	30: // Parse results
		_intRet := STRING_TO_INT(_inst_strRet);
		IF _intRet > 0 THEN
			_bResult := TRUE;
			THIS^.M_LogMessage(_strEND_MSG);
			// DO ANY PARSING HERE
			bConnected := TRUE;
		// Set error if command failed
		ELSE
			THIS^.M_SetError(_udintERROR_ID, _strERROR_MSG);
		END_IF
		// Go back to start
		_inst_intStep := 0;
END_CASE
M_StartMarking := _bResult;
intMStartMarkingStep := _inst_intStep;
END_METHOD

METHOD PUBLIC M_StopMarking : BOOL
VAR_INPUT
END_VAR

VAR CONSTANT
	_strCOMMAND_NAME : T_MaxString	:= 'StopMarking'; // Name of the API method
	_timeCOMMAND_TIMEOUT : TIME		:= T#30S; // Max time to receive API response
	_strSTART_MSG : T_MaxString		:= 'StoppingMarking'; // Prints when method starts
	_strEND_MSG : T_MaxString		:= 'StoppedMarking'; // Prints when method finishes
	_udintERROR_ID : UDINT			:= KeyenceLaserMarkerMDX2000_Error.FailedToStopMarking; // Error ID to set if command fails
	_strERROR_MSG : T_MaxString		:= 'Failed to Stop Marking by Laser Marker!'; // Error message to set if command fails
END_VAR

VAR_INST
	_inst_arrParams: T_ApiParameterList; // Parameters array
	_inst_arrOutputs: T_ApiParameterList; // Outputs array
	_inst_strRet: T_ApiParamValue; // Return string from the router
	_inst_intStep: INT; // Current method step
	_inst_fbParams: FB_ApiParamBuilder; // Parameter builder FB
END_VAR

VAR
	_bComplete: BOOL; // True if the routing finishes
	_intRet: INT; // Return string converted to an integer
	_bResult : BOOL; // Output of the method
END_VAR
_bResult := FALSE;
bMStopMarkingBusy := TRUE;
_inst_intStep := intMStopMarkingStep;
CASE _inst_intStep OF
	0: // Wait for no error and router not busy
		IF NOT THIS^.P_bError AND NOT bRouterBusy THEN
			bRouterBusy := TRUE;
			_inst_intStep := _inst_intStep + 10;
		END_IF
		
	10: // Initialize parameters
		THIS^.M_LogMessage(_strSTART_MSG);
		_inst_fbParams.M_ClearParameters();
		// ADD ANY PARAMETERS HERE
		_inst_fbParams.M_OutputToParameterList(_inst_arrParams);
		_inst_intStep := _inst_intStep + 10;
		
	20: // Route the command
		_bComplete := M_RouterHelper(
			_in_strMethodName := _strCOMMAND_NAME, 
			_in_timeTimeout := _timeCOMMAND_TIMEOUT,
			_inout_arrParams := _inst_arrParams,
			_inout_arrOutputs := _inst_arrOutputs,
			_out_strReturnValue=>_inst_strRet);
		
		// If route completed, move to next step
		IF _bComplete THEN
			_inst_intStep := _inst_intStep + 10;
			bRouterBusy := FALSE;
		ELSIF THIS^.P_bError THEN
			_inst_intStep := 0;
			bRouterBusy := FALSE;
		END_IF
		
	30: // Parse results
		_intRet := STRING_TO_INT(_inst_strRet);
		IF _intRet > 0 THEN
			_bResult := TRUE;
			THIS^.M_LogMessage(_strEND_MSG);
			// DO ANY PARSING HERE
			bConnected := TRUE;
		// Set error if command failed
		ELSE
			THIS^.M_SetError(_udintERROR_ID, _strERROR_MSG);
		END_IF
		// Go back to start
		_inst_intStep := 0;
END_CASE
M_StopMarking := _bResult;
intMStopMarkingStep := _inst_intStep;
END_METHOD

METHOD M_UpdateAllMarkingInformation : BOOL
VAR_INPUT
	MaxNumberOfBlocks	: INT;
//	MarkingInfo_Array	: ARRAY [0..255] OF OneBlockInfo;
END_VAR

VAR CONSTANT
	_strCOMMAND_NAME : T_MaxString	:= 'UpdateAllMarkingInformation'; // Name of the API method
	_timeCOMMAND_TIMEOUT : TIME		:= T#30S; // Max time to receive API response
	_strSTART_MSG : T_MaxString		:= 'UpdatingAllMarkingInformationInTheLaserProgram'; // Prints when method starts
	_strEND_MSG : T_MaxString		:= 'UpdatedAllMarkingInformationInTheLaserProgram'; // Prints when method finishes
	_udintERROR_ID : UDINT			:= KeyenceLaserMarkerMDX2000_Error.FailedToUpdateAllMarkingInformation; // Error ID to set if command fails
	_strERROR_MSG : T_MaxString		:= 'Failed to update All Marking Information in the Laser Marker program!'; // Error message to set if command fails
END_VAR

VAR_INST
	_inst_arrParams: T_ApiParameterList; // Parameters array
	_inst_arrOutputs: T_ApiParameterList; // Outputs array
	_inst_strRet: T_ApiParamValue; // Return string from the router
	_inst_intStep: INT; // Current method step
	_inst_fbParams: FB_ApiParamBuilder; // Parameter builder FB
END_VAR

VAR
	_bComplete: BOOL; // True if the routing finishes
	_intRet: INT; // Return string converted to an integer
	_bResult : BOOL; // Output of the method
	intIndex: INT;
	intIndex2 : INT;
	bOneTimeOnly : BOOL := TRUE;
END_VAR
_bResult := FALSE;
bMUpdateAllMarkingInfoBusy := TRUE;
_inst_intStep := intMUpdateAllMarkingInfoStep;
CASE _inst_intStep OF
	0: // Wait for no error and router not busy
		IF NOT THIS^.P_bError AND NOT bRouterBusy THEN
			bRouterBusy := TRUE;
			_inst_intStep := _inst_intStep + 10;
		END_IF
		
	10: // Initialize parameters
		THIS^.M_LogMessage(_strSTART_MSG);
		_inst_fbParams.M_ClearParameters();
		// ADD ANY PARAMETERS HERE
		_inst_fbParams.M_AddParameter('MaxNumberOfBlocks', MaxNumberOfBlocks);
		_inst_fbParams.M_OutputToParameterList(_inst_arrParams);
		_inst_intStep := _inst_intStep + 10;
		
	20: // Route the command
		_bComplete := M_RouterHelper(
			_in_strMethodName := _strCOMMAND_NAME, 
			_in_timeTimeout := _timeCOMMAND_TIMEOUT,
			_inout_arrParams := _inst_arrParams,
			_inout_arrOutputs := _inst_arrOutputs,
			_out_strReturnValue=>_inst_strRet);
		
		// If route completed, move to next step
		IF _bComplete THEN
			_inst_intStep := _inst_intStep + 10;
			bRouterBusy := FALSE;
		ELSIF THIS^.P_bError THEN
			_inst_intStep := 0;
			bRouterBusy := FALSE;
		END_IF
		
	30: // Parse results
		_intRet := STRING_TO_INT(_inst_strRet);
		IF _intRet > 0 THEN
			_bResult := TRUE;
			THIS^.M_LogMessage(_strEND_MSG);
			// DO ANY PARSING HERE
			_inst_fbParams.M_LoadFromParameterList(_inst_arrOutputs);
			bConnected := TRUE;
		// Set error if command failed
		ELSE
			THIS^.M_SetError(_udintERROR_ID, _strERROR_MSG);
		END_IF
		// Go back to start
		_inst_intStep := 0;
END_CASE
M_UpdateAllMarkingInformation := _bResult;
intMUpdateAllMarkingInfoStep := _inst_intStep;
END_METHOD

METHOD PUBLIC M_UpdateSingleBlockMarkingInformation : BOOL
VAR_INPUT
	BlockNumber : INT;
	BlockData : STRING;
	MarkEnabled : BOOL;
END_VAR

VAR CONSTANT
	_strCOMMAND_NAME : T_MaxString	:= 'UpdateSingleBlockMarkingInformation'; // Name of the API method
	_timeCOMMAND_TIMEOUT : TIME		:= T#30S; // Max time to receive API response
	_strSTART_MSG : T_MaxString		:= 'UpdatingSingleBlockMarkingInformationInTheLaserProgram'; // Prints when method starts
	_strEND_MSG : T_MaxString		:= 'UpdatedSingleBlockMarkingInformationInTheLaserProgram'; // Prints when method finishes
	_udintERROR_ID : UDINT			:= KeyenceLaserMarkerMDX2000_Error.FailedToUpdateSingleBlockMarkingInformation; // Error ID to set if command fails
	_strERROR_MSG : T_MaxString		:= 'Failed to update single block Marking Information in the Laser Marker program!'; // Error message to set if command fails
END_VAR

VAR_INST
	_inst_arrParams: T_ApiParameterList; // Parameters array
	_inst_arrOutputs: T_ApiParameterList; // Outputs array
	_inst_strRet: T_ApiParamValue; // Return string from the router
	_inst_intStep: INT; // Current method step
	_inst_fbParams: FB_ApiParamBuilder; // Parameter builder FB
END_VAR

VAR
	_bComplete: BOOL; // True if the routing finishes
	_intRet: INT; // Return string converted to an integer
	_bResult : BOOL; // Output of the method
	BlockType_INT : INT;
END_VAR
_bResult := FALSE;
bMUpdateSingleBlockInfoBusy := TRUE;
_inst_intStep := intMUpdateSingleBlockInfoStep;
CASE _inst_intStep OF
	0: // Wait for no error and router not busy
		IF NOT THIS^.P_bError AND NOT bRouterBusy THEN
			bRouterBusy := TRUE;
			_inst_intStep := _inst_intStep + 10;
		END_IF
		
	10: // Initialize parameters
		THIS^.M_LogMessage(_strSTART_MSG);
		_inst_fbParams.M_ClearParameters();
		// ADD ANY PARAMETERS HERE
		_inst_fbParams.M_AddParameter('BlockNumber', BlockNumber);
		_inst_fbParams.M_AddParameter('BlockData', BlockData);
		_inst_fbParams.M_AddParameter('MarkEnabled', MarkEnabled);
		_inst_fbParams.M_OutputToParameterList(_inst_arrParams);
		_inst_intStep := _inst_intStep + 10;
		
	20: // Route the command
		_bComplete := M_RouterHelper(
			_in_strMethodName := _strCOMMAND_NAME, 
			_in_timeTimeout := _timeCOMMAND_TIMEOUT,
			_inout_arrParams := _inst_arrParams,
			_inout_arrOutputs := _inst_arrOutputs,
			_out_strReturnValue=>_inst_strRet);
		
		// If route completed, move to next step
		IF _bComplete THEN
			_inst_intStep := _inst_intStep + 10;
			bRouterBusy := FALSE;
		ELSIF THIS^.P_bError THEN
			_inst_intStep := 0;
			bRouterBusy := FALSE;
		END_IF
		
	30: // Parse results
		_intRet := STRING_TO_INT(_inst_strRet);
		IF _intRet > 0 THEN
			_bResult := TRUE;
			THIS^.M_LogMessage(_strEND_MSG);
			// DO ANY PARSING HERE
			_inst_fbParams.M_LoadFromParameterList(_inst_arrOutputs);
			bConnected := TRUE;
		// Set error if command failed
		ELSE
			THIS^.M_SetError(_udintERROR_ID, _strERROR_MSG);
		END_IF
		// Go back to start
		_inst_intStep := 0;
END_CASE
M_UpdateSingleBlockMarkingInformation := _bResult;
intMUpdateSingleBlockInfoStep := _inst_intStep;
END_METHOD

(* This method should explicitly get the current program loaded on the device.
	If the current program is successfully gotten, this method should return
	TRUE and set P_strCurrentProgram and strCurrentProgram to the gotten
	program name. If this method fails, both should be set to empty strings. *)
METHOD M_GetCurrentProgram : BOOL
VAR_OUTPUT
	(* This should be set to the name of the currently loaded program if
		the method was successful, or a blank string otherwise. *)
	strCurrentProgram	: Sensata_Common.T_MaxString;
END_VAR
VAR CONSTANT
	_strCOMMAND_NAME : T_MaxString	:= 'GetCurrentProgram'; // Name of the API method
	_timeCOMMAND_TIMEOUT : TIME		:= T#45S; // Max time to receive API response
	_strSTART_MSG : T_MaxString		:= 'GettingCurrentProgramFromLaserMemory'; // Prints when method starts
	_strEND_MSG : T_MaxString		:= 'GotCurrentProgramFromLaserMemory'; // Prints when method finishes
	_udintERROR_ID : UDINT			:= KeyenceLaserMarkerMDX2000_Error.FailedToGetCurrentProgram; // Error ID to set if command fails
	_strERROR_MSG : T_MaxString		:= 'Failed to Get Current Laser Program from Laser Marker!'; // Error message to set if command fails
END_VAR

VAR_INST
	_inst_arrParams: T_ApiParameterList; // Parameters array
	_inst_arrOutputs: T_ApiParameterList; // Outputs array
	_inst_strRet: T_ApiParamValue; // Return string from the router
	_inst_intStep: INT; // Current method step
	_inst_fbParams: FB_ApiParamBuilder; // Parameter builder FB
END_VAR

VAR
	_bComplete: BOOL; // True if the routing finishes
	_intRet: INT; // Return string converted to an integer
	_bResult : BOOL; // Output of the method
END_VAR
_bResult := FALSE;
bMGetCurrentProgBusy := TRUE;
_inst_intStep := intMGetCurrentProgStep;
CASE _inst_intStep OF
	0: // Wait for no error and router not busy
		IF NOT THIS^.P_bError AND NOT bRouterBusy THEN
			bRouterBusy := TRUE;
			_inst_intStep := _inst_intStep + 10;
		END_IF
		
	10: // Initialize parameters
		THIS^.M_LogMessage(_strSTART_MSG);
		_inst_fbParams.M_ClearParameters();
		// ADD ANY PARAMETERS HERE
		_inst_fbParams.M_OutputToParameterList(_inst_arrParams);
		_inst_intStep := _inst_intStep + 10;
		
	20: // Route the command
		_bComplete := M_RouterHelper(
			_in_strMethodName := _strCOMMAND_NAME, 
			_in_timeTimeout := _timeCOMMAND_TIMEOUT,
			_inout_arrParams := _inst_arrParams,
			_inout_arrOutputs := _inst_arrOutputs,
			_out_strReturnValue=>_inst_strRet);
		
		// If route completed, move to next step
		IF _bComplete THEN
			_inst_intStep := _inst_intStep + 10;
			bRouterBusy := FALSE;
		ELSIF THIS^.P_bError THEN
			_inst_intStep := 0;
			bRouterBusy := FALSE;
		END_IF
		
	30: // Parse results
		_intRet := STRING_TO_INT(_inst_strRet);
		IF _intRet > 0 THEN
			_bResult := TRUE;
			THIS^.M_LogMessage(_strEND_MSG);
			// DO ANY PARSING HERE
			_inst_fbParams.M_LoadFromParameterList(_inst_arrOutputs);
			strCurrentProgram := _inst_fbParams.M_ParseString(_inst_fbParams.M_GetParameter('programName'));
			bConnected := TRUE;
		// Set error if command failed
		ELSE
			THIS^.M_SetError(_udintERROR_ID, _strERROR_MSG);
		END_IF
		// Go back to start
		_inst_intStep := 0;
END_CASE
M_GetCurrentProgram := _bResult;
intMGetCurrentProgStep := _inst_intStep;
END_METHOD

(* This method should explicitly check the program state of the device.
	Once the program state is known, this method should return TRUE and set
	P_enumProgramState and enumProgramState to the relevant E_ProgramState
	value, else it should set both to E_ProgramState.Unknown. *)
METHOD M_GetProgramState : BOOL
VAR_OUTPUT
	(* If the program state is successfully gotten, this should be set to
		the relevant E_ProgramState value. If this method fails, this should
		be set to E_ProgramState.Unknown. *)
	enumProgramState	: Sensata_Common.E_ProgramState;
END_VAR
M_GetProgramState := TRUE;
THIS^.M_LogWarning('M_GetProgramState is not implemented!');
END_METHOD

(* This method should load a new program onto the device, and then return TRUE
	once program loading is completed. Once this method begins the program loading
	process, P_strCurrentProgram should be cleared unless it is still explicitly
	known to be loaded. *)
METHOD M_LoadProgram : BOOL
VAR_INPUT
	(* String representing the program to load. If string must be in a specific
		format, make sure to override this comment to document it. *)
	//strProgram	: Sensata_Common.T_MaxString;
	
	//Replace filepath with just program number and also 
//	filepath : STRING;	// filepath where the program is stored
//	LaserMemoryLocation : INT; // Laser Memory location where the program needs to be loaded 
	
END_VAR

VAR CONSTANT
	_strCOMMAND_NAME : T_MaxString	:= 'LoadProgram'; // Name of the API method
	_timeCOMMAND_TIMEOUT : TIME		:= T#30S; // Max time to receive API response
	_strSTART_MSG : T_MaxString		:= 'LoadingProgramToLaser'; // Prints when method starts
	_strEND_MSG : T_MaxString		:= 'ProgramLoadedToLaser'; // Prints when method finishes
	_udintERROR_ID : UDINT			:= KeyenceLaserMarkerMDX2000_Error.FailedToSendProgramToLaser; // Error ID to set if command fails
	_strERROR_MSG : T_MaxString		:= 'Failed to Load Program to Laser Marker!'; // Error message to set if command fails
END_VAR

VAR_INST
	_inst_arrParams: T_ApiParameterList; // Parameters array
	_inst_arrOutputs: T_ApiParameterList; // Outputs array
	_inst_strRet: T_ApiParamValue; // Return string from the router
	_inst_intStep: INT; // Current method step
	_inst_fbParams: FB_ApiParamBuilder; // Parameter builder FB
END_VAR

VAR
	_bComplete: BOOL; // True if the routing finishes
	_intRet: INT; // Return string converted to an integer
	_bResult : BOOL; // Output of the method	
END_VAR
_bResult := FALSE;
bMLoadProgramBusy := TRUE;
_inst_intStep := intMLoadProgramStep;
CASE _inst_intStep OF
	0: // Wait for no error and router not busy
		IF NOT THIS^.P_bError AND NOT bRouterBusy THEN
			bRouterBusy := TRUE;
			_inst_intStep := _inst_intStep + 10;
		END_IF
		
	10: // Initialize parameters
		THIS^.M_LogMessage(_strSTART_MSG);
		_inst_fbParams.M_ClearParameters();
		// ADD ANY PARAMETERS HERE
		_inst_fbParams.M_AddParameter('programName', in_strProgram);
		_inst_fbParams.M_OutputToParameterList(_inst_arrParams);
		_inst_intStep := _inst_intStep + 10;
		
	20: // Route the command
		_bComplete := M_RouterHelper(
			_in_strMethodName := _strCOMMAND_NAME, 
			_in_timeTimeout := _timeCOMMAND_TIMEOUT,
			_inout_arrParams := _inst_arrParams,
			_inout_arrOutputs := _inst_arrOutputs,
			_out_strReturnValue=>_inst_strRet);
		
		// If route completed, move to next step
		IF _bComplete THEN
			_inst_intStep := _inst_intStep + 10;
			bRouterBusy := FALSE;
		ELSIF THIS^.P_bError THEN
			_inst_intStep := 0;
			bRouterBusy := FALSE;
		END_IF
		
	30: // Parse results
		_intRet := STRING_TO_INT(_inst_strRet);
		IF _intRet > 0 THEN
			_bResult := TRUE;
			THIS^.M_LogMessage(_strEND_MSG);
			// DO ANY PARSING HERE
		// Set error if command failed
		ELSE
			THIS^.M_SetError(_udintERROR_ID, _strERROR_MSG);
		END_IF
		// Go back to start
		_inst_intStep := 0;
END_CASE
M_LoadProgram := _bResult;
intMLoadProgramStep := _inst_intStep;
END_METHOD

(* This program should move to the program state from whatever state it was in
	to the Paused state, and then return TRUE once successful. If the program
	state is Stopped, this method should return TRUE but keep the current state
	as Stopped, since Paused at the beginning at the program is equivalent to
	being Stopped. *)
METHOD M_PauseProgram : BOOL
M_PauseProgram := TRUE;
THIS^.M_LogWarning('M_PauseProgram is not implemented!');
END_METHOD

METHOD PUBLIC M_SaveCurrentLaserProgramtoPC : BOOL
VAR_INPUT
	LaserProgramFolderPath : STRING;
END_VAR
VAR_OUTPUT
	out_bool_SaveProgramToPC_Success : BOOL;
END_VAR
VAR CONSTANT
	_strCOMMAND_NAME : T_MaxString	:= 'SaveCurrentLaserProgramToPC'; // Name of the API method
	_timeCOMMAND_TIMEOUT : TIME		:= T#45S; // Max time to receive API response
	_strSTART_MSG : T_MaxString		:= 'SavingCurrentProgram'; // Prints when method starts
	_strEND_MSG : T_MaxString		:= 'SavedCurrentProgram'; // Prints when method finishes
	_udintERROR_ID : UDINT			:= KeyenceLaserMarkerMDX2000_Error.FailedToSaveCurrentLaserProgramToPC; // Error ID to set if command fails
	_strERROR_MSG : T_MaxString		:= 'Failed to Save Current Laser Program to PC from Laser Marker!'; // Error message to set if command fails
END_VAR

VAR_INST
	_inst_arrParams: T_ApiParameterList; // Parameters array
	_inst_arrOutputs: T_ApiParameterList; // Outputs array
	_inst_strRet: T_ApiParamValue; // Return string from the router
	_inst_intStep: INT; // Current method step
	_inst_fbParams: FB_ApiParamBuilder; // Parameter builder FB
END_VAR

VAR
	_bComplete: BOOL; // True if the routing finishes
	_intRet: INT; // Return string converted to an integer
	_bResult : BOOL; // Output of the method
END_VAR
_bResult := FALSE;
bMSaveCurrentLaserProgramtoPCBusy := TRUE;
_inst_intStep := intMSaveCurrentLaserProgramtoPC;
CASE _inst_intStep OF
	0: // Wait for no error and router not busy
		IF NOT THIS^.P_bError AND NOT bRouterBusy THEN
			bRouterBusy := TRUE;
			_inst_intStep := _inst_intStep + 10;
		END_IF
		
	10: // Initialize parameters
		THIS^.M_LogMessage(_strSTART_MSG);
		_inst_fbParams.M_ClearParameters();
		// ADD ANY PARAMETERS HERE
		_inst_fbParams.M_AddParameter('LaserProgramFolderPath',LaserProgramFolderPath);
		_inst_fbParams.M_OutputToParameterList(_inst_arrParams);
		_inst_intStep := _inst_intStep + 10;
		
	20: // Route the command
		_bComplete := M_RouterHelper(
			_in_strMethodName := _strCOMMAND_NAME, 
			_in_timeTimeout := _timeCOMMAND_TIMEOUT,
			_inout_arrParams := _inst_arrParams,
			_inout_arrOutputs := _inst_arrOutputs,
			_out_strReturnValue=>_inst_strRet);
		
		// If route completed, move to next step
		IF _bComplete THEN
			_inst_intStep := _inst_intStep + 10;
			bRouterBusy := FALSE;
		ELSIF THIS^.P_bError THEN
			_inst_intStep := 0;
			bRouterBusy := FALSE;
		END_IF
		
	30: // Parse results
		_intRet := STRING_TO_INT(_inst_strRet);
		IF _intRet > 0 THEN
			_bResult := TRUE;
			THIS^.M_LogMessage(_strEND_MSG);
			// DO ANY PARSING HERE
			_inst_fbParams.M_LoadFromParameterList(_inst_arrOutputs);
			out_bool_SaveProgramToPC_Success := _inst_fbParams.M_ParseBool(_inst_fbParams.M_GetParameter('out_bool_SaveProgramToPC_Success'));
			bConnected := TRUE;
		// Set error if command failed
		ELSE
			THIS^.M_SetError(_udintERROR_ID, _strERROR_MSG);
		END_IF
		// Go back to start
		_inst_intStep := 0;
END_CASE
M_SaveCurrentLaserProgramtoPC := _bResult;
intMSaveCurrentLaserProgramtoPC := _inst_intStep;
END_METHOD

METHOD PUBLIC M_SendProgramtoLaser : BOOL
VAR_INPUT
	filepath : STRING;	// filepath where the program is stored
	LaserMemoryLocation : INT; // Laser Memory location where the program needs to be loaded 
END_VAR

VAR_OUTPUT
	out_bool_SendProgramToLaserSuccess : BOOL;
END_VAR

VAR CONSTANT
	_strCOMMAND_NAME : T_MaxString	:= 'SendProgramtoLaser'; // Name of the API method
	_timeCOMMAND_TIMEOUT : TIME		:= T#30S; // Max time to receive API response
	_strSTART_MSG : T_MaxString		:= 'SendingProgramToLaser'; // Prints when method starts
	_strEND_MSG : T_MaxString		:= 'SentProgramToLaser'; // Prints when method finishes
	_udintERROR_ID : UDINT			:= KeyenceLaserMarkerMDX2000_Error.FailedToSendProgramToLaser; // Error ID to set if command fails
	_strERROR_MSG : T_MaxString		:= 'Failed to Send Program to Laser Marker!'; // Error message to set if command fails
END_VAR

VAR_INST
	_inst_arrParams: T_ApiParameterList; // Parameters array
	_inst_arrOutputs: T_ApiParameterList; // Outputs array
	_inst_strRet: T_ApiParamValue; // Return string from the router
	_inst_intStep: INT; // Current method step
	_inst_fbParams: FB_ApiParamBuilder; // Parameter builder FB
END_VAR

VAR
	_bComplete: BOOL; // True if the routing finishes
	_intRet: INT; // Return string converted to an integer
	_bResult : BOOL; // Output of the method	

END_VAR
_bResult := FALSE;
bMSendProgramToLaserBusy := TRUE;
_inst_intStep := intMSendProgramToLaserStep;
CASE _inst_intStep OF
	0: // Wait for no error and router not busy
		IF NOT THIS^.P_bError AND NOT bRouterBusy THEN
			bRouterBusy := TRUE;
			_inst_intStep := _inst_intStep + 10;
		END_IF
		
	10: // Initialize parameters
		THIS^.M_LogMessage(_strSTART_MSG);
		_inst_fbParams.M_ClearParameters();
		// ADD ANY PARAMETERS HERE
		_inst_fbParams.M_AddParameter('filepath', filepath);
		_inst_fbParams.M_AddParameter('LaserMemoryLocation', LaserMemoryLocation);
		_inst_fbParams.M_OutputToParameterList(_inst_arrParams);
		_inst_intStep := _inst_intStep + 10;
		
	20: // Route the command
		_bComplete := M_RouterHelper(
			_in_strMethodName := _strCOMMAND_NAME, 
			_in_timeTimeout := _timeCOMMAND_TIMEOUT,
			_inout_arrParams := _inst_arrParams,
			_inout_arrOutputs := _inst_arrOutputs,
			_out_strReturnValue=>_inst_strRet);
		
		// If route completed, move to next step
		IF _bComplete THEN
			_inst_intStep := _inst_intStep + 10;
			bRouterBusy := FALSE;
		ELSIF THIS^.P_bError THEN
			_inst_intStep := 0;
			bRouterBusy := FALSE;
		END_IF
		
	30: // Parse results
		_intRet := STRING_TO_INT(_inst_strRet);
		IF _intRet > 0 THEN
			_bResult := TRUE;
			THIS^.M_LogMessage(_strEND_MSG);
			// DO ANY PARSING HERE
			_inst_fbParams.M_LoadFromParameterList(_inst_arrOutputs);
			out_bool_SendProgramToLaserSuccess := _inst_fbParams.M_ParseBool(_inst_fbParams.M_GetParameter('out_bool_SendProgramToLaserSuccess'));
			bConnected := TRUE;
		// Set error if command failed
		ELSE
			THIS^.M_SetError(_udintERROR_ID, _strERROR_MSG);
		END_IF
		// Go back to start
		_inst_intStep := 0;
END_CASE
M_SendProgramtoLaser := _bResult;
intMSendProgramToLaserStep := _inst_intStep;
END_METHOD

(* This should move the program state from whatever state it is in to the
	Running state, and then return TRUE once successful. Starting from the
	Paused state should always continue execution from whatever point the
	program was at when the program was initially paused. *)
METHOD M_StartProgram : BOOL
M_StartProgram := TRUE;
THIS^.M_LogWarning('M_StartProgram is not implemented!');
END_METHOD

(* This should change the program state from whatever state it was in to the
	Stopped state and then return TRUE. Moving to the Stopped state should
	always reset the program execution back to the beginning. *)
METHOD M_StopProgram : BOOL
M_StopProgram := TRUE;
THIS^.M_LogWarning('M_StopProgram is not implemented!');
END_METHOD

METHOD PUBLIC M_UpdateSingleProgramBlockData : BOOL
VAR_INPUT
	LaserProgramMemoryLocation : INT;
	BlockNumber : INT;
	BlockData : STRING;
	BlockType : BlockTypes;
END_VAR
VAR_OUTPUT
	out_bool_UpdateData_Success : BOOL;
END_VAR
VAR CONSTANT
	_strCOMMAND_NAME : T_MaxString	:= 'UpdateSingleBlockData'; // Name of the API method
	_timeCOMMAND_TIMEOUT : TIME		:= T#30S; // Max time to receive API response
	_strSTART_MSG : T_MaxString		:= 'UpdatingSingleBlockdataInTheLaserProgram'; // Prints when method starts
	_strEND_MSG : T_MaxString		:= 'UpdatedSingleBlockdataInTheLaserProgram'; // Prints when method finishes
	_udintERROR_ID : UDINT			:= KeyenceLaserMarkerMDX2000_Error.FailedToUpdateSingleBlockData; // Error ID to set if command fails
	_strERROR_MSG : T_MaxString		:= 'Failed to update single block data in the Laser Marker program!'; // Error message to set if command fails
END_VAR

VAR_INST
	_inst_arrParams: T_ApiParameterList; // Parameters array
	_inst_arrOutputs: T_ApiParameterList; // Outputs array
	_inst_strRet: T_ApiParamValue; // Return string from the router
	_inst_intStep: INT; // Current method step
	_inst_fbParams: FB_ApiParamBuilder; // Parameter builder FB
END_VAR

VAR
	_bComplete: BOOL; // True if the routing finishes
	_intRet: INT; // Return string converted to an integer
	_bResult : BOOL; // Output of the method
	BlockType_INT : INT;
END_VAR
_bResult := FALSE;
bMUpdateSingleProgramBlockDataBusy := TRUE;
_inst_intStep := intMUpdateSingleProgramBlockDataStep;
CASE _inst_intStep OF
	0: // Wait for no error and router not busy
		IF NOT THIS^.P_bError AND NOT bRouterBusy THEN
			bRouterBusy := TRUE;
			_inst_intStep := _inst_intStep + 10;
		END_IF
		
	10: // Initialize parameters
		THIS^.M_LogMessage(_strSTART_MSG);
		_inst_fbParams.M_ClearParameters();
		// ADD ANY PARAMETERS HERE
		BlockType_INT := TO_INT(BlockType);
		_inst_fbParams.M_AddParameter('LaserProgramMemoryLocation', LaserProgramMemoryLocation);
		_inst_fbParams.M_AddParameter('BlockNumber', BlockNumber);
		_inst_fbParams.M_AddParameter('BlockData', BlockData);
		_inst_fbParams.M_AddParameter('BlockType', BlockType_INT);
		_inst_fbParams.M_OutputToParameterList(_inst_arrParams);
		_inst_intStep := _inst_intStep + 10;
		
	20: // Route the command
		_bComplete := M_RouterHelper(
			_in_strMethodName := _strCOMMAND_NAME, 
			_in_timeTimeout := _timeCOMMAND_TIMEOUT,
			_inout_arrParams := _inst_arrParams,
			_inout_arrOutputs := _inst_arrOutputs,
			_out_strReturnValue=>_inst_strRet);
		
		// If route completed, move to next step
		IF _bComplete THEN
			_inst_intStep := _inst_intStep + 10;
			bRouterBusy := FALSE;
		ELSIF THIS^.P_bError THEN
			_inst_intStep := 0;
			bRouterBusy := FALSE;
		END_IF
		
	30: // Parse results
		_intRet := STRING_TO_INT(_inst_strRet);
		IF _intRet > 0 THEN
			_bResult := TRUE;
			THIS^.M_LogMessage(_strEND_MSG);
			// DO ANY PARSING HERE
			_inst_fbParams.M_LoadFromParameterList(_inst_arrOutputs);
			out_bool_UpdateData_Success := _inst_fbParams.M_ParseBool(_inst_fbParams.M_GetParameter('out_bool_UpdateData_Success'));
			bConnected := TRUE;
		// Set error if command failed
		ELSE
			THIS^.M_SetError(_udintERROR_ID, _strERROR_MSG);
		END_IF
		// Go back to start
		_inst_intStep := 0;
END_CASE
M_UpdateSingleProgramBlockData := _bResult;
intMUpdateSingleProgramBlockDataStep := _inst_intStep;
END_METHOD

METHOD PUBLIC M_UpdateSingleProgramBlockMarkEnabled : BOOL
VAR_INPUT
	LaserProgramMemoryLocation : INT;
	BlockNumber : INT;
	BlockType : BlockTypes;
	MarkEnabled : BOOL;
	//int LaserProgramMemoryLocation, int BlockNumber, bool MarkEnabled, BlockTypes BlockType, out bool out_bool_UpdateSingleBlockMarkEnabledIntheLaser_Success
END_VAR
VAR_OUTPUT
	out_bool_MarkEnabled_Success : BOOL;
END_VAR
VAR CONSTANT
	_strCOMMAND_NAME : T_MaxString	:= 'UpdateSingleBlockMarkEnabled'; // Name of the API method
	_timeCOMMAND_TIMEOUT : TIME		:= T#30S; // Max time to receive API response
	_strSTART_MSG : T_MaxString		:= 'UpdatingSingleBlockMarkEnabledStatusInTheLaserProgram'; // Prints when method starts
	_strEND_MSG : T_MaxString		:= 'UpdatedSingleBlockMarkEnabledStatusInTheLaserProgram'; // Prints when method finishes
	_udintERROR_ID : UDINT			:= KeyenceLaserMarkerMDX2000_Error.FailedToUpdateSingleBlockMarkEnabledProperty; // Error ID to set if command fails
	_strERROR_MSG : T_MaxString		:= 'Failed to update single block mark enabled status in the Laser Marker program!'; // Error message to set if command fails
END_VAR

VAR_INST
	_inst_arrParams: T_ApiParameterList; // Parameters array
	_inst_arrOutputs: T_ApiParameterList; // Outputs array
	_inst_strRet: T_ApiParamValue; // Return string from the router
	_inst_intStep: INT; // Current method step
	_inst_fbParams: FB_ApiParamBuilder; // Parameter builder FB
END_VAR

VAR
	_bComplete: BOOL; // True if the routing finishes
	_intRet: INT; // Return string converted to an integer
	_bResult : BOOL; // Output of the method
	_dummy_pointer : PVOID;
	BlockType_INT : INT;
END_VAR
_bResult := FALSE;
bMUpdateSingleProgramBlockMarkingEnabledBusy := TRUE;
_inst_intStep := intMUpdateSingleProgramBlockMarkingEnabledStep;
CASE _inst_intStep OF
	0: // Wait for no error and router not busy
		IF NOT THIS^.P_bError AND NOT bRouterBusy THEN
			bRouterBusy := TRUE;
			_inst_intStep := _inst_intStep + 10;
		END_IF
		
	10: // Initialize parameters
		THIS^.M_LogMessage(_strSTART_MSG);
		_inst_fbParams.M_ClearParameters();
		// ADD ANY PARAMETERS HERE
		BlockType_INT := TO_INT(BlockType);
		_inst_fbParams.M_AddParameter('LaserProgramMemoryLocation', LaserProgramMemoryLocation);
		_inst_fbParams.M_AddParameter('BlockNumber', BlockNumber);
		_inst_fbParams.M_AddParameter('MarkEnabled', MarkEnabled);
		_inst_fbParams.M_AddParameter('BlockType', BlockType_INT);
		_inst_fbParams.M_OutputToParameterList(_inst_arrParams);
		_inst_intStep := _inst_intStep + 10;
		
	20: // Route the command
		_bComplete := M_RouterHelper(
			_in_strMethodName := _strCOMMAND_NAME, 
			_in_timeTimeout := _timeCOMMAND_TIMEOUT,
			_inout_arrParams := _inst_arrParams,
			_inout_arrOutputs := _inst_arrOutputs,
			_out_strReturnValue=>_inst_strRet);
		
		// If route completed, move to next step
		IF _bComplete THEN
			_inst_intStep := _inst_intStep + 10;
			bRouterBusy := FALSE;
		ELSIF THIS^.P_bError THEN
			_inst_intStep := 0;
			bRouterBusy := FALSE;
		END_IF
		
	30: // Parse results
		_intRet := STRING_TO_INT(_inst_strRet);
		IF _intRet > 0 THEN
			_bResult := TRUE;
			THIS^.M_LogMessage(_strEND_MSG);
			// DO ANY PARSING HERE
			_inst_fbParams.M_LoadFromParameterList(_inst_arrOutputs);
			out_bool_MarkEnabled_Success := _inst_fbParams.M_ParseBool(_inst_fbParams.M_GetParameter('out_bool_MarkEnabled_Success'));
			bConnected := TRUE;
		// Set error if command failed
		ELSE
			THIS^.M_SetError(_udintERROR_ID, _strERROR_MSG);
		END_IF
		// Go back to start
		_inst_intStep := 0;
END_CASE
M_UpdateSingleProgramBlockMarkEnabled := _bResult;
intMUpdateSingleProgramBlockMarkingEnabledStep := _inst_intStep;
END_METHOD

(* This property should be TRUE while any method in this interface is actively
	executing, or FALSE otherwise. *)
PROPERTY P_bProgramControlBusy : BOOL
GET
END_GET
END_PROPERTY

(* The current E_ProgramState value of the device. This should be reset to
	E_ProgramState.Unknown if any methods in this interface interact with the
	device but fail. *)
PROPERTY P_enumProgramState : Sensata_Common.E_ProgramState
GET
END_GET
END_PROPERTY

(* The value of the currently loaded program. This should only be set by
	M_LoadProgram or M_GetCurrentProgram, and set to a blank string if either
	fail. *)
PROPERTY P_strCurrentProgram : Sensata_Common.T_MaxString
GET
END_GET
END_PROPERTY

METHOD PUBLIC M_GetLaserActivatedStatus : BOOL
VAR_INPUT
//	LaserProgramFolderPath : STRING;
END_VAR
VAR_OUTPUT
	out_IsLaserActivated : BOOL;
END_VAR
VAR CONSTANT
	_strCOMMAND_NAME : T_MaxString	:= 'GetLaserActivatedStatus'; // Name of the API method
	_timeCOMMAND_TIMEOUT : TIME		:= T#30S; // Max time to receive API response
	_strSTART_MSG : T_MaxString		:= 'GettingLaserActivatedStatus'; // Prints when method starts
	_strEND_MSG : T_MaxString		:= 'ReceivedLaserActivatedStatus'; // Prints when method finishes
	_udintERROR_ID : UDINT			:= KeyenceLaserMarkerMDX2000_Error.FailedToGetLaserActivatedStatus; // Error ID to set if command fails
	_strERROR_MSG : T_MaxString		:= 'Failed to Get Laser Activated Status from Laser Marker!'; // Error message to set if command fails
END_VAR

VAR_INST
	_inst_arrParams: T_ApiParameterList; // Parameters array
	_inst_arrOutputs: T_ApiParameterList; // Outputs array
	_inst_strRet: T_ApiParamValue; // Return string from the router
	_inst_intStep: INT; // Current method step
	_inst_fbParams: FB_ApiParamBuilder; // Parameter builder FB
END_VAR

VAR
	_bComplete: BOOL; // True if the routing finishes
	_intRet: INT; // Return string converted to an integer
	_bResult : BOOL; // Output of the method
END_VAR
_bResult := FALSE;
bMGetLaserActivatedStatusBusy := TRUE;
_inst_intStep := intMGetLaserActivatedStatusStep;
CASE _inst_intStep OF
	0: // Wait for no error and router not busy
		IF NOT THIS^.P_bError AND NOT bRouterBusy THEN
			bRouterBusy := TRUE;
			_inst_intStep := _inst_intStep + 10;
		END_IF
		
	10: // Initialize parameters
		THIS^.M_LogMessage(_strSTART_MSG);
		_inst_fbParams.M_ClearParameters();
		// ADD ANY PARAMETERS HERE
		_inst_fbParams.M_OutputToParameterList(_inst_arrParams);
		_inst_intStep := _inst_intStep + 10;
		
	20: // Route the command
		_bComplete := M_RouterHelper(
			_in_strMethodName := _strCOMMAND_NAME, 
			_in_timeTimeout := _timeCOMMAND_TIMEOUT,
			_inout_arrParams := _inst_arrParams,
			_inout_arrOutputs := _inst_arrOutputs,
			_out_strReturnValue=>_inst_strRet);
		
		// If route completed, move to next step
		IF _bComplete THEN
			_inst_intStep := _inst_intStep + 10;
			bRouterBusy := FALSE;
		ELSIF THIS^.P_bError THEN
			_inst_intStep := 0;
			bRouterBusy := FALSE;
		END_IF
		
	30: // Parse results
		_intRet := STRING_TO_INT(_inst_strRet);
		IF _intRet > 0 THEN
			_bResult := TRUE;
			THIS^.M_LogMessage(_strEND_MSG);
			// DO ANY PARSING HERE
			_inst_fbParams.M_LoadFromParameterList(_inst_arrOutputs);
			out_IsLaserActivated := _inst_fbParams.M_ParseBool(_inst_fbParams.M_GetParameter('out_IsLaserActivated'));
			bConnected := TRUE;
		// Set error if command failed
		ELSE
			THIS^.M_SetError(_udintERROR_ID, _strERROR_MSG);
		END_IF
		// Go back to start
		_inst_intStep := 0;
END_CASE
M_GetLaserActivatedStatus := _bResult;
intMGetLaserActivatedStatusStep := _inst_intStep;
END_METHOD

METHOD PUBLIC M_GetLaserErrorStatus : BOOL
VAR_INPUT
//	LaserProgramFolderPath : STRING;
END_VAR
VAR_OUTPUT
	out_bool_IsLaserError : BOOL;
END_VAR
VAR CONSTANT
	_strCOMMAND_NAME : T_MaxString	:= 'GetLaserErrorStatus'; // Name of the API method
	_timeCOMMAND_TIMEOUT : TIME		:= T#30S; // Max time to receive API response
	_strSTART_MSG : T_MaxString		:= 'GettingLaserErrorStatus'; // Prints when method starts
	_strEND_MSG : T_MaxString		:= 'ReceivedLaserErrorStatus'; // Prints when method finishes
	_udintERROR_ID : UDINT			:= KeyenceLaserMarkerMDX2000_Error.FailedToGetLaserErrorStatus; // Error ID to set if command fails
	_strERROR_MSG : T_MaxString		:= 'Failed to Get Laser Error Status from Laser Marker!'; // Error message to set if command fails
END_VAR

VAR_INST
	_inst_arrParams: T_ApiParameterList; // Parameters array
	_inst_arrOutputs: T_ApiParameterList; // Outputs array
	_inst_strRet: T_ApiParamValue; // Return string from the router
	_inst_intStep: INT; // Current method step
	_inst_fbParams: FB_ApiParamBuilder; // Parameter builder FB
END_VAR

VAR
	_bComplete: BOOL; // True if the routing finishes
	_intRet: INT; // Return string converted to an integer
	_bResult : BOOL; // Output of the method
END_VAR
_bResult := FALSE;
bMGetLaserErrorStatusBusy := TRUE;
_inst_intStep := intMGetLaserErrorStatusStep;
CASE _inst_intStep OF
	0: // Wait for no error and router not busy
		IF NOT THIS^.P_bError AND NOT bRouterBusy THEN
			bRouterBusy := TRUE;
			_inst_intStep := _inst_intStep + 10;
		END_IF
		
	10: // Initialize parameters
		THIS^.M_LogMessage(_strSTART_MSG);
		_inst_fbParams.M_ClearParameters();
		// ADD ANY PARAMETERS HERE
		_inst_fbParams.M_OutputToParameterList(_inst_arrParams);
		_inst_intStep := _inst_intStep + 10;
		
	20: // Route the command
		_bComplete := M_RouterHelper(
			_in_strMethodName := _strCOMMAND_NAME, 
			_in_timeTimeout := _timeCOMMAND_TIMEOUT,
			_inout_arrParams := _inst_arrParams,
			_inout_arrOutputs := _inst_arrOutputs,
			_out_strReturnValue=>_inst_strRet);
		
		// If route completed, move to next step
		IF _bComplete THEN
			_inst_intStep := _inst_intStep + 10;
			bRouterBusy := FALSE;
		ELSIF THIS^.P_bError THEN
			_inst_intStep := 0;
			bRouterBusy := FALSE;
		END_IF
		
	30: // Parse results
		_intRet := STRING_TO_INT(_inst_strRet);
		IF _intRet > 0 THEN
			_bResult := TRUE;
			THIS^.M_LogMessage(_strEND_MSG);
			// DO ANY PARSING HERE
			_inst_fbParams.M_LoadFromParameterList(_inst_arrOutputs);
			out_bool_IsLaserError := _inst_fbParams.M_ParseBool(_inst_fbParams.M_GetParameter('out_bool_IsLaserError'));
			bConnected := TRUE;
		// Set error if command failed
		ELSE
			THIS^.M_SetError(_udintERROR_ID, _strERROR_MSG);
		END_IF
		// Go back to start
		_inst_intStep := 0;
END_CASE
M_GetLaserErrorStatus := _bResult;
intMGetLaserErrorStatusStep := _inst_intStep;
END_METHOD

METHOD PUBLIC M_GetLaserMarkingStatus : BOOL
VAR_INPUT

END_VAR
VAR_OUTPUT
	out_bool_IsLaserMarking : BOOL;
END_VAR
VAR CONSTANT
	_strCOMMAND_NAME : T_MaxString	:= 'GetLaserMarkingStatus'; // Name of the API method
	_timeCOMMAND_TIMEOUT : TIME		:= T#30S; // Max time to receive API response
	_strSTART_MSG : T_MaxString		:= 'GettingLaserMarkingStatus'; // Prints when method starts
	_strEND_MSG : T_MaxString		:= 'ReceivedLaserMarkingStatus'; // Prints when method finishes
	_udintERROR_ID : UDINT			:= KeyenceLaserMarkerMDX2000_Error.FailedToGetLaserMarkingStatus; // Error ID to set if command fails
	_strERROR_MSG : T_MaxString		:= 'Failed to Get Laser Marking Status from Laser Marker!'; // Error message to set if command fails
END_VAR

VAR_INST
	_inst_arrParams: T_ApiParameterList; // Parameters array
	_inst_arrOutputs: T_ApiParameterList; // Outputs array
	_inst_strRet: T_ApiParamValue; // Return string from the router
	_inst_intStep: INT; // Current method step
	_inst_fbParams: FB_ApiParamBuilder; // Parameter builder FB
END_VAR

VAR
	_bComplete: BOOL; // True if the routing finishes
	_intRet: INT; // Return string converted to an integer
	_bResult : BOOL; // Output of the method
END_VAR
_bResult := FALSE;
bMGetLaserMarkingStatusBusy := TRUE;
_inst_intStep := intMGetLaserMarkingStatusStep;
CASE _inst_intStep OF
	0: // Wait for no error and router not busy
		IF NOT THIS^.P_bError AND NOT bRouterBusy THEN
			bRouterBusy := TRUE;
			_inst_intStep := _inst_intStep + 10;
		END_IF
		
	10: // Initialize parameters
		THIS^.M_LogMessage(_strSTART_MSG);
		_inst_fbParams.M_ClearParameters();
		// ADD ANY PARAMETERS HERE
		_inst_fbParams.M_OutputToParameterList(_inst_arrParams);
		_inst_intStep := _inst_intStep + 10;
		
	20: // Route the command
		_bComplete := M_RouterHelper(
			_in_strMethodName := _strCOMMAND_NAME, 
			_in_timeTimeout := _timeCOMMAND_TIMEOUT,
			_inout_arrParams := _inst_arrParams,
			_inout_arrOutputs := _inst_arrOutputs,
			_out_strReturnValue=>_inst_strRet);
		
		// If route completed, move to next step
		IF _bComplete THEN
			_inst_intStep := _inst_intStep + 10;
			bRouterBusy := FALSE;
		ELSIF THIS^.P_bError THEN
			_inst_intStep := 0;
			bRouterBusy := FALSE;
		END_IF
		
	30: // Parse results
		_intRet := STRING_TO_INT(_inst_strRet);
		IF _intRet > 0 THEN
			_bResult := TRUE;
			THIS^.M_LogMessage(_strEND_MSG);
			// DO ANY PARSING HERE
			_inst_fbParams.M_LoadFromParameterList(_inst_arrOutputs);
			out_bool_IsLaserMarking := _inst_fbParams.M_ParseBool(_inst_fbParams.M_GetParameter('out_bool_IsLaserMarking'));
			bConnected := TRUE;
		// Set error if command failed
		ELSE
			THIS^.M_SetError(_udintERROR_ID, _strERROR_MSG);
		END_IF
		// Go back to start
		_inst_intStep := 0;
END_CASE
M_GetLaserMarkingStatus := _bResult;
intMGetLaserMarkingStatusStep := _inst_intStep;
END_METHOD

METHOD PUBLIC M_GetLaserStatus : BOOL
VAR_INPUT

END_VAR
VAR_OUTPUT
	out_string_laserStatus : STRING;
END_VAR
VAR CONSTANT
	_strCOMMAND_NAME : T_MaxString	:= 'GetLaserStatus'; // Name of the API method
	_timeCOMMAND_TIMEOUT : TIME		:= T#30S; // Max time to receive API response
	_strSTART_MSG : T_MaxString		:= 'GettingLaserStatus'; // Prints when method starts
	_strEND_MSG : T_MaxString		:= 'GotLaserStatus'; // Prints when method finishes
	_udintERROR_ID : UDINT			:= KeyenceLaserMarkerMDX2000_Error.FailedToGetLaserStatus; // Error ID to set if command fails
	_strERROR_MSG : T_MaxString		:= 'Failed to Get Laser Status from Laser Marker!'; // Error message to set if command fails
END_VAR

VAR_INST
	_inst_arrParams: T_ApiParameterList; // Parameters array
	_inst_arrOutputs: T_ApiParameterList; // Outputs array
	_inst_strRet: T_ApiParamValue; // Return string from the router
	_inst_intStep: INT; // Current method step
	_inst_fbParams: FB_ApiParamBuilder; // Parameter builder FB
END_VAR

VAR
	_bComplete: BOOL; // True if the routing finishes
	_intRet: INT; // Return string converted to an integer
	_bResult : BOOL; // Output of the method
END_VAR
_bResult := FALSE;
bMGetLaserStatusBusy := TRUE;
_inst_intStep := intMGetLaserStatusStep;
CASE _inst_intStep OF
	0: // Wait for no error and router not busy
		IF NOT THIS^.P_bError AND NOT bRouterBusy THEN
			bRouterBusy := TRUE;
			_inst_intStep := _inst_intStep + 10;
		END_IF
		
	10: // Initialize parameters
		THIS^.M_LogMessage(_strSTART_MSG);
		_inst_fbParams.M_ClearParameters();
		// ADD ANY PARAMETERS HERE
		_inst_fbParams.M_OutputToParameterList(_inst_arrParams);
		_inst_intStep := _inst_intStep + 10;
		
	20: // Route the command
		_bComplete := M_RouterHelper(
			_in_strMethodName := _strCOMMAND_NAME, 
			_in_timeTimeout := _timeCOMMAND_TIMEOUT,
			_inout_arrParams := _inst_arrParams,
			_inout_arrOutputs := _inst_arrOutputs,
			_out_strReturnValue=>_inst_strRet);
		
		// If route completed, move to next step
		IF _bComplete THEN
			_inst_intStep := _inst_intStep + 10;
			bRouterBusy := FALSE;
		ELSIF THIS^.P_bError THEN
			_inst_intStep := 0;
			bRouterBusy := FALSE;
		END_IF
		
	30: // Parse results
		_intRet := STRING_TO_INT(_inst_strRet);
		IF _intRet > 0 THEN
			_bResult := TRUE;
			THIS^.M_LogMessage(_strEND_MSG);
			// DO ANY PARSING HERE
			_inst_fbParams.M_LoadFromParameterList(_inst_arrOutputs);
			out_string_laserStatus := _inst_fbParams.M_ParseString(_inst_fbParams.M_GetParameter('_out_string_laserStatus'));
			bConnected := TRUE;
		// Set error if command failed
		ELSE
			THIS^.M_SetError(_udintERROR_ID, _strERROR_MSG);
		END_IF
		// Go back to start
		_inst_intStep := 0;
END_CASE
M_GetLaserStatus := _bResult;
intMGetLaserStatusStep := _inst_intStep;
END_METHOD

(* This should clear any errors on the device and bring it to a state where
	it is ready to be energized or otherwise activated. *)
METHOD M_Reset : BOOL
VAR CONSTANT
	_strCOMMAND_NAME : T_MaxString	:= 'Reset'; // Name of the API method
	_timeCOMMAND_TIMEOUT : TIME		:= T#30S; // Max time to receive API response
	_strSTART_MSG : T_MaxString		:= 'Resetting'; // Prints when method starts
	_strEND_MSG : T_MaxString		:= 'Reset'; // Prints when method finishes
	_udintERROR_ID : UDINT			:= KeyenceLaserMarkerMDX2000_Error.FailedToReset; // Error ID to set if command fails
	_strERROR_MSG : T_MaxString		:= 'Failed to reset laser!'; // Error message to set if command fails
	_udintAPI_ERR_ID : UDINT		:= KeyenceLaserMarkerMDX2000_Error.CommandRouterError; // Error to set if there is an error on the API block
	_strAPI_ERR_MSG : T_MaxString	:= 'Error while trying to get API connect status!'; // Error message to set if there is an error on the API block
END_VAR
VAR_INST
	_inst_arrParams: T_ApiParameterList; // Parameters array
	_inst_arrOutputs: T_ApiParameterList; // Outputs array
	_inst_strRet: T_ApiParamValue; // Return string from the router
	_inst_intStep: INT; // Current step
	_inst_fbParams: FB_ApiParamBuilder; // Parameter builder FB
END_VAR
VAR
	_intRet: INT; // Return string converted to an integer
	_bComplete: BOOL; // True if the routing finishes
	_bGotStatus: BOOL; // Goes true once connect status is received
	_bApiConnected: BOOL; // True if API is connected
	_bResult : BOOL; // Output of the method
END_VAR
_bResult := FALSE;
bMResetBusy := TRUE;
_inst_intStep := intMResetStep;
CASE _inst_intStep OF
	0: // Clear errors
		THIS^.M_ClearError();
		in_fbApi.M_ClearError();
		bResetBusy := TRUE;
		_inst_intStep := _inst_intStep + 10;
		
	10: // Check connection status
		_bGotStatus := in_fbApi.M_GetConnectStatus(bConnected => _bApiConnected);
		IF _bGotStatus THEN
			// If the API is connected, go to the next step
			IF _bApiConnected THEN
				_inst_intStep := _inst_intStep + 10;
			// If the API is not connected, reset is done
			ELSE
				_inst_intStep := 0;
				M_Reset := TRUE;
				THIS^.M_LogMessage(_strEND_MSG);
			END_IF
			
		// Set an error 
		ELSIF in_fbApi.P_bError THEN
			_inst_intStep := 0;
			THIS^.M_SetError(_udintAPI_ERR_ID, _strAPI_ERR_MSG);
		END_IF
		
	20: // Wait for router to be free
		IF NOT bRouterBusy THEN
			_inst_intStep := _inst_intStep + 10;
			bRouterBusy := TRUE;
		END_IF
		
	30: // Setup parameters for reset command
		THIS^.M_LogMessage(_strSTART_MSG);
		_inst_fbParams.M_ClearParameters();
		_inst_fbParams.M_OutputToParameterList(_inst_arrParams);
		_inst_intStep := _inst_intStep + 10;
		
	40: // Route command
		_bComplete := M_RouterHelper(
			_in_strMethodName := _strCOMMAND_NAME, 
			_in_timeTimeout := _timeCOMMAND_TIMEOUT,
			_inout_arrParams := _inst_arrParams,
			_inout_arrOutputs := _inst_arrOutputs,
			_out_strReturnValue=>_inst_strRet);
		
		// If route completed, parse results
		IF _bComplete THEN
			_inst_intStep := _inst_intStep + 10;
			bRouterBusy := FALSE;
		ELSIF THIS^.P_bError THEN
			_inst_intStep := 0;
			bRouterBusy := FALSE;
			bResetBusy := FALSE;
		END_IF
		
	50: // Parse results

		// If return value is greater than 1 then robot was reset
		_intRet := STRING_TO_INT(_inst_strRet);
		IF _intRet > 0 THEN
			_bResult := TRUE;
			THIS^.M_LogMessage(_strEND_MSG);
			
		// Else robot failed to reset
		ELSE
			THIS^.M_SetError(_udintERROR_ID, _strERROR_MSG);
		END_IF
		
		// Back to start
		_inst_intStep := 0;
		bResetBusy := FALSE;
END_CASE
M_Reset := _bResult;
intMResetStep := _inst_intStep;
END_METHOD

(* This property should be TRUE while any method in this interface is actively
	executing, or FALSE otherwise. *)
PROPERTY P_bResetBusy : BOOL
GET
END_GET
END_PROPERTY

ACTION A_CommandRecovery:
IF NOT bRouterHelperBusy AND intRouterHelperStep > 0 THEN
	intRouterHelperStep := 0;
	THIS^.M_LogWarning('Router helper ended prematurely!');
END_IF
bRouterHelperBusy := FALSE;

IF NOT bMConnectBusy AND intMConnectStep > 0 THEN
	bRouterBusy := FALSE;
	intMConnectStep := 0;
	THIS^.M_LogWarning('Connect ended prematurely!');
END_IF
bMConnectBusy := FALSE;

IF NOT bMDisconnectBusy AND intMDisconnectStep > 0 THEN
	bRouterBusy := FALSE;
	intMDisconnectStep := 0;
	THIS^.M_LogWarning('Disconnect ended prematurely!');
END_IF
bMDisconnectBusy := FALSE;

IF NOT bMGetConnectStatusBusy AND intMGetConnectStatusStep > 0 THEN
	bRouterBusy := FALSE;
	intMGetConnectStatusStep := 0;
	THIS^.M_LogWarning('Get Connect Status ended prematurely!');
END_IF
bMGetConnectStatusBusy := FALSE;

IF NOT bMPeakCurrentProgramBusy AND intMPeakCurrentProgramStep > 0 THEN
	bRouterBusy := FALSE;
	intMPeakCurrentProgramStep := 0;
	THIS^.M_LogWarning('Peak Current Program ended prematurely!');
END_IF
bMPeakCurrentProgramBusy := FALSE;

IF NOT bMSendMarkingParamsBusy AND intMSendMarkingParamsStep > 0 THEN
	bRouterBusy := FALSE;
	intMSendMarkingParamsStep := 0;
	THIS^.M_LogWarning('Send Marking Params ended prematurely!');
END_IF
bMSendMarkingParamsBusy := FALSE;

IF NOT bMStartMarkingBusy AND intMStartMarkingStep > 0 THEN
	bRouterBusy := FALSE;
	intMStartMarkingStep := 0;
	THIS^.M_LogWarning('Start Marking ended prematurely!');
END_IF
bMStartMarkingBusy := FALSE;

IF NOT bMStopMarkingBusy AND intMStopMarkingStep > 0 THEN
	bRouterBusy := FALSE;
	intMStopMarkingStep := 0;
	THIS^.M_LogWarning('Stop Marking ended prematurely!');
END_IF
bMStopMarkingBusy := FALSE;

IF NOT bMUpdateAllMarkingInfoBusy AND intMUpdateAllMarkingInfoStep > 0 THEN
	bRouterBusy := FALSE;
	intMUpdateAllMarkingInfoStep := 0;
	THIS^.M_LogWarning('Update All Marking Info ended prematurely!');
END_IF
bMUpdateAllMarkingInfoBusy := FALSE;

IF NOT bMUpdateSingleBlockInfoBusy AND intMUpdateSingleBlockInfoStep > 0 THEN
	bRouterBusy := FALSE;
	intMUpdateSingleBlockInfoStep := 0;
	THIS^.M_LogWarning('Update Single Block Info ended prematurely!');
END_IF
bMUpdateSingleBlockInfoBusy := FALSE;

IF NOT bMGetCurrentProgBusy AND intMGetCurrentProgStep > 0 THEN
	bRouterBusy := FALSE;
	intMGetCurrentProgStep := 0;
	THIS^.M_LogWarning('Get Current Program ended prematurely!');
END_IF
bMGetCurrentProgBusy := FALSE;

IF NOT bMLoadProgramBusy AND intMLoadProgramStep > 0 THEN
	bRouterBusy := FALSE;
	intMLoadProgramStep := 0;
	THIS^.M_LogWarning('Load Program ended prematurely!');
END_IF
bMLoadProgramBusy := FALSE;

IF NOT bMSaveCurrentLaserProgramtoPCBusy AND intMSaveCurrentLaserProgramtoPC > 0 THEN
	bRouterBusy := FALSE;
	intMSaveCurrentLaserProgramtoPC := 0;
	THIS^.M_LogWarning('Save Current Laser Program to PC ended prematurely!');
END_IF
bMSaveCurrentLaserProgramtoPCBusy := FALSE;

IF NOT bMSendProgramToLaserBusy AND intMSendProgramToLaserStep > 0 THEN
	bRouterBusy := FALSE;
	intMSendProgramToLaserStep := 0;
	THIS^.M_LogWarning('Send Program to Laser ended prematurely!');
END_IF
bMSendProgramToLaserBusy := FALSE;

IF NOT bMStartProgramBusy AND intMStartProgramStep > 0 THEN
	bRouterBusy := FALSE;
	intMStartProgramStep := 0;
	THIS^.M_LogWarning('Start Program ended prematurely!');
END_IF
bMStartProgramBusy := FALSE;

IF NOT bMUpdateSingleProgramBlockDataBusy AND intMUpdateSingleProgramBlockDataStep > 0 THEN
	bRouterBusy := FALSE;
	intMUpdateSingleProgramBlockDataStep := 0;
	THIS^.M_LogWarning('Update Single Program Block Data ended prematurely!');
END_IF
bMUpdateSingleProgramBlockDataBusy := FALSE;

IF NOT bMUpdateSingleProgramBlockMarkingEnabledBusy AND intMUpdateSingleProgramBlockMarkingEnabledStep > 0 THEN
	bRouterBusy := FALSE;
	intMUpdateSingleProgramBlockMarkingEnabledStep := 0;
	THIS^.M_LogWarning('Update Single Program Block Marking Enabled ended prematurely!');
END_IF
bMUpdateSingleProgramBlockMarkingEnabledBusy := FALSE;

IF NOT bMGetLaserActivatedStatusBusy AND intMGetLaserActivatedStatusStep > 0 THEN
	bRouterBusy := FALSE;
	intMGetLaserActivatedStatusStep := 0;
	THIS^.M_LogWarning('Get Laser Activated Status ended prematurely!');
END_IF
bMGetLaserActivatedStatusBusy := FALSE;

IF NOT bMGetLaserErrorStatusBusy AND intMGetLaserErrorStatusStep > 0 THEN
	bRouterBusy := FALSE;
	intMGetLaserErrorStatusStep := 0;
	THIS^.M_LogWarning('Get Laser Error Status ended prematurely!');
END_IF
bMGetLaserErrorStatusBusy := FALSE;

IF NOT bMGetLaserMarkingStatusBusy AND intMGetLaserMarkingStatusStep > 0 THEN
	bRouterBusy := FALSE;
	intMGetLaserMarkingStatusStep := 0;
	THIS^.M_LogWarning('Get Laser Marking Status ended prematurely!');
END_IF
bMGetLaserMarkingStatusBusy := FALSE;

IF NOT bMGetLaserStatusBusy AND intMGetLaserStatusStep > 0 THEN
	bRouterBusy := FALSE;
	intMGetLaserStatusStep := 0;
	THIS^.M_LogWarning('Get Laser Status ended prematurely!');
END_IF
bMGetLaserStatusBusy := FALSE;

IF NOT bMClearErrorBusy AND intMClearErrorStep > 0 THEN
	bRouterBusy := FALSE;
	intMClearErrorStep := 0;
	THIS^.M_LogWarning('Clear Error ended prematurely!');
END_IF
bMClearErrorBusy := FALSE;

IF NOT bMResetBusy AND intMResetStep > 0 THEN
	bRouterBusy := FALSE;
	intMResetStep := 0;
	THIS^.M_LogWarning('Reset ended prematurely!');
END_IF
bMResetBusy := FALSE;
END_ACTION

(*
Sends the given method to the API and receives and partially parses the result.
*)
METHOD PRIVATE M_RouterHelper : BOOL
VAR_INPUT
	(* Name of the method to call. *)
	_in_strMethodName : T_MaxString;
	(* Maximum time to wait for method response. *)
	_in_timeTimeout : TIME;
END_VAR
VAR_IN_OUT
	(* The array of parameters to send to the API. *)
	_inout_arrParams : T_ApiParameterList;
	(* The array that gets populated with any method output data. *)
	_inout_arrOutputs : T_ApiParameterList;
END_VAR
VAR_OUTPUT
	(* JSON string of the method return value. *)
	_out_strReturnValue: T_ApiParamValue;
END_VAR
VAR_INST
	(* Current step. *)
	_inst_intStep: INT;
	(* True if the method executed. *)
	_inst_bExec: BOOL;
	(* Return string of the method. *)
	_inst_strRet: T_ApiParamValue;
END_VAR
VAR
	(* True once the command routing finishes. *)
	_bComplete: BOOL;
	(* True once the API connects. *)
	_bApiConnect: BOOL;
END_VAR
bRouterHelperBusy := TRUE;
_inst_intStep := intRouterHelperStep;
CASE _inst_intStep OF
	0: // Start process only if there is no error on this FB
		IF NOT THIS^.P_bError THEN
			in_fbApi.M_ClearError();
			_inst_intStep := 10;
		END_IF
		
	10: // Check if command router connected
		IF NOT in_fbApi.P_bConnected THEN
			_inst_intStep := 20; // Go to API connect step
		ELSE
			_inst_intStep := 30; // Go to route command step
		END_IF
		
	20: // Connect the command router
		_bApiConnect := in_fbApi.M_Connect();
		IF _bApiConnect THEN
			_inst_intStep := _inst_intStep + 10; // Go to next step
		ELSIF in_fbApi.P_bError THEN
			THIS^.M_SetError(KeyenceLaserMarkerMDX2000_Error.CommandRouterError, 'Error on command router function block while connecting!');
			_inst_intStep := 0; // Go back to start
		END_IF
		
	30:	// Route the command
		_bComplete := in_fbApi.M_RouteCommand(
			_in_strModuleId := in_strUniqueId,
			_in_strMethodName := _in_strMethodName,
			_in_timeTimeout := _in_timeTimeout,
			_inout_arrParameters := _inout_arrParams,
			_inout_arrOutputs := _inout_arrOutputs,
			_out_bCommandExecuted => _inst_bExec,
			_out_strReturnValue => _inst_strRet);
		IF _bComplete THEN
			_inst_intStep := _inst_intStep + 10; // Go to next step
		ELSIF in_fbApi.P_bError THEN
			THIS^.M_SetError(KeyenceLaserMarkerMDX2000_Error.CommandRouterError, 'Error on command router function block while routing command!');
			_inst_intStep := 0; // Go back to start
		END_IF
		
	40: // Check result then go back to start
		IF NOT _inst_bExec THEN
			THIS^.M_SetError(KeyenceLaserMarkerMDX2000_Error.CommandFault, 'Method in API failed to execute!');
		ELSE
			_out_strReturnValue := _inst_strRet;
			M_RouterHelper := TRUE;
		END_IF
		_inst_intStep := 0; // Go back to start
END_CASE
intRouterHelperStep := _inst_intStep;
END_METHOD

END_FUNCTION_BLOCK

// Project Information/F_GetCompany
// This function has been automatically generated from the project information.
{attribute 'signature_flag' := '1073741824'}
{attribute 'TcGenerated'}
{attribute 'no-analysis'}
FUNCTION F_GetCompany : WSTRING
VAR_INPUT
	
END_VAR

F_GetCompany := "Sensata Technologies";

END_FUNCTION

// Project Information/F_GetTitle
// This function has been automatically generated from the project information.
{attribute 'signature_flag' := '1073741824'}
{attribute 'TcGenerated'}
{attribute 'no-analysis'}
FUNCTION F_GetTitle : WSTRING
VAR_INPUT
	
END_VAR

F_GetTitle := "Sensata_Laser";

END_FUNCTION

// Project Information/F_GetVersion
// This function has been automatically generated from the project information.
{attribute 'signature_flag' := '1073741824'}
{attribute 'TcGenerated'}
{attribute 'no-analysis'}
FUNCTION F_GetVersion : ST_LibVersion
VAR_INPUT
	
END_VAR

F_GetVersion.iMajor := 0;
F_GetVersion.iMinor := 0;
F_GetVersion.iBuild := 1;
F_GetVersion.iRevision := 0;
F_GetVersion.sVersion := '0.0.1';
F_GetVersion.nFlags := 0;

END_FUNCTION
